FUNCTION_BLOCK FB_autoStore EXTENDS FB_Generic
VAR_INPUT
END_VAR
VAR_OUTPUT
END_VAR
VAR
	lamp			: BOOL;	
	eStates			: E_AutoStore_States := E_AutoStore_States.IDLE;;
	eStateTemp		: E_AutoStore_States := E_AutoStore_States.IDLE;
	
	mcAxis_lift 			: FB_MotionAxis_MC;
	st_mcAxis_lift 			: ST_MotionAxis_MC;
	AxisRef_lift			: AXIS_REF;
	
	mcAxis_transfer 		: FB_MotionAxis_MC;
	st_mcAxis_transfer		: ST_MotionAxis_MC;
	AxisRef_transfer		: AXIS_REF;
	
	door_closed						: BOOL;
	button_start					: BOOL;	
	button_stop						: BOOL;	
	sensor_lift_atDownPos			: BOOL;
	sensor_transfer_atWorkingPos	: BOOL;
	sensor_transfer_atFeedingPos	: BOOL;
	
	bUpStairs						: BOOL;
	bExchangeTote					: BOOL;
	
	
	autostore_status	: AutostoreStatus;
END_VAR	
VAR PERSISTENT
	rPos_lift_up				: REAL;//340
	rPos_lift_down				: REAL;
	rPos_transfer_feeding		: REAL;
	rPos_transfer_working		: REAL;//636	
END_VAR

SUPER^();
IF sInstanceName='autoStore_1' THEN
	rPos_lift_up				:= 350;
	rPos_lift_down				:= 0;
	rPos_transfer_feeding		:= 0;
	rPos_transfer_working		:= 656;	
END_IF
IF sInstanceName='autoStore_2' THEN
	rPos_lift_up				:= 350;
	rPos_lift_down				:= 0;
	rPos_transfer_feeding		:= 0;
	rPos_transfer_working		:= 624;	
END_IF
IF sInstanceName='autoStore_1' THEN
	IF NOT subscribed THEN
		GVL.PubSubService.Subscribe(E_Topics.AUTOSTORE1_EXCHANGE,sInstanceName,THIS^);
		subscribed	:= TRUE;
	END_IF
END_IF
IF sInstanceName='autoStore_2' THEN
	IF NOT subscribed THEN
		GVL.PubSubService.Subscribe(E_Topics.AUTOSTORE2_EXCHANGE,sInstanceName,THIS^);
		subscribed	:= TRUE;
	END_IF
END_IF

//sComponent_name		:= _sInstanceName;
//iComponetID			:= ModuleID.SAMPLE1;

infoLevel	:= ServerityLevelType.WARNING;

(*
Description: 
the callback that will be invoked when there is a publish for what the subscriber was subscribed to.
*)
METHOD Callback
VAR_INPUT
	data : PubSubData;
END_VAR
IF door_closed THEN
	IF sInstanceName='autoStore_1' THEN
		CASE data.Topic OF
			E_Topics.AUTOSTORE1_EXCHANGE:
				IF autostore_status<>AutostoreStatus.EXCHANGING THEN
					bExchangeTote	:= TRUE;	
				END_IF
		END_CASE	
	END_IF
	IF sInstanceName='autoStore_2' THEN
		CASE data.Topic OF
			E_Topics.AUTOSTORE2_EXCHANGE:
				IF autostore_status<>AutostoreStatus.EXCHANGING THEN
					bExchangeTote	:= TRUE;	
				END_IF		
		END_CASE	
	END_IF
END_IF
END_METHOD

{attribute 'object_name' := 'M_Aborting'}
METHOD M_Aborting
CASE fbUnitModeManager.eModeStatus OF	
	ePMLProtUnitMode_Production, ePMLProtUnitMode_Manual:		

		st_mcAxis_lift.mcMoveAbsolute.Execute		:= FALSE;
		st_mcAxis_lift.mcStop.Execute				:= TRUE;	
		st_mcAxis_transfer.mcMoveAbsolute.Execute	:= FALSE;
		st_mcAxis_transfer.mcStop.Execute			:= TRUE;
		iAging_test	:= 0;
		M_StateComplete();
			
	ePMLProtUnitMode_Maintenance, ePMLUnitMode_Service:
		
		M_StateComplete();
END_CASE
END_METHOD

METHOD M_agingTest : BOOL
VAR_INPUT
	rVelocity_percent	: REAL;
END_VAR
END_METHOD

{attribute 'object_name' := 'M_Completing'}
METHOD M_Completing
CASE fbUnitModeManager.eModeStatus OF
	ePMLProtUnitMode_Production:
		;
END_CASE
END_METHOD

{attribute 'object_name' := 'M_Execute'}
METHOD M_Execute
IF door_closed THEN
	st_mcAxis_transfer.mcStop.Execute	:= FALSE;
	st_mcAxis_lift.mcStop.Execute		:= FALSE;
	st_mcAxis_transfer.mcReset.Execute	:= TRUE;
	st_mcAxis_lift.mcReset.Execute		:= TRUE;	
ELSE
	st_mcAxis_transfer.mcStop.Execute	:= TRUE;
	st_mcAxis_lift.mcStop.Execute		:= TRUE;
	RETURN;
END_IF
CASE fbUnitModeManager.eModeStatus OF
	ePMLProtUnitMode_Production:		//Mode Production
//////////////////////////////////////////////////////////timeout//////////////////////////////////////////	
		iStateTemp	:= eStateTemp;
		ton_timeout();
		IF eStateTemp=eStates THEN
			ton_timeout.IN	:=TRUE;
		ELSE
			ton_timeout.IN	:=FALSE;
			eStateTemp	:= eStates;	
			M_Log(eLogType:=ServerityLevelType.INFO,sTextLog:='');
			IF ton_timeout.Q THEN
				RETURN;
			END_IF
		END_IF
		IF ton_timeout.Q THEN	
			ton_timeout.IN	:=FALSE;
			CASE eStates OF	
				E_AutoStore_States.ERROR:	
					alarm_temp.Message	:= GenerateErrorMsg(errorType:='M',iState := iStateTemp,errorMsg:='in error state.');
				ELSE
				alarm_temp.Message	:= GenerateErrorMsg(errorType:='M',iState := iStateTemp,errorMsg:='time out');
			END_CASE
//////////////////////////////////////////////////////////states don't want to timeout and trig error//////////////////////////////////////////				
			IF 	eStates<>E_AutoStore_States.IDLE AND
				eStates<>E_AutoStore_States.WAIT AND
				eStates<>E_AutoStore_States.WAIT_CMD
			THEN 
				IF sInstanceName='autoStore_1' THEN
					GVL.pml_adminAlarm.M_SetAlarm(stAdmin:=GVL.PackTags1.Admin,stAlarm:=alarm_temp);
				END_IF
				IF sInstanceName='autoStore_2' THEN
					GVL.pml_adminAlarm.M_SetAlarm(stAdmin:=GVL.PackTags2.Admin,stAlarm:=alarm_temp);
				END_IF					
			END_IF
		END_IF
//////////////////////////////////////////////////////////auto running process//////////////////////////////////////////			
		CASE eStates OF 
				E_AutoStore_States.IDLE:
					ton_timeout.PT	:= T#1MS;						
					eStates	:= E_AutoStore_States.INIT;				
				E_AutoStore_States.INIT:
					ton_timeout.PT	:= T#1S;
					st_mcAxis_transfer.mcMoveAbsolute.Execute	:= FALSE;
					st_mcAxis_lift.mcMoveAbsolute.Execute	:= FALSE;
					autostore_status	:= AutostoreStatus.UNKNOWN;
					eStates	:= E_AutoStore_States.WAIT; 
				E_AutoStore_States.WAIT:
					ton_timeout.PT	:= T#10S;
					eStates	:= E_AutoStore_States.WAIT_CMD; 
				E_AutoStore_States.WAIT_CMD:
					IF bExchangeTote OR button_start THEN
						bExchangeTote	:= FALSE;
						autostore_status	:= AutostoreStatus.EXCHANGING;
						eStates	:= E_AutoStore_States.LIFT_MOVE_DOWN;
					END_IF
				////////////////////////////lift move down///////////////////////////////////		
				E_AutoStore_States.LIFT_MOVE_DOWN:	
					st_mcAxis_lift.mcMoveAbsolute.Execute	:= TRUE;					
					st_mcAxis_lift.rActualPosSet	:= rPos_lift_down;
					st_mcAxis_lift.rVelocitySet		:= 400;					
					IF st_mcAxis_lift.mcMoveAbsolute.Done THEN
						st_mcAxis_lift.mcMoveAbsolute.Execute	:= FALSE;
						eStates	:= E_AutoStore_States.LIFT_DOWN_SENSOR_DETECTED;
					END_IF
				E_AutoStore_States.LIFT_DOWN_SENSOR_DETECTED:	
					IF TRUE OR sensor_lift_atDownPos THEN
						IF bUpStairs THEN
							eStates	:= E_AutoStore_States.TRANSFER_MOVE_FEEDING;
							bUpStairs	:= FALSE;
						ELSE
							eStates	:= E_AutoStore_States.TRANSFER_MOVE_WORKING;
							bUpStairs	:= TRUE;
						END_IF					
					END_IF
				////////////////////////////upstairs///////////////////////////////////	
				E_AutoStore_States.TRANSFER_MOVE_FEEDING:	
					st_mcAxis_transfer.mcMoveAbsolute.Execute	:= TRUE;					
					st_mcAxis_transfer.rActualPosSet	:= rPos_transfer_feeding;
					st_mcAxis_transfer.rVelocitySet		:= 600;					
					IF st_mcAxis_transfer.mcMoveAbsolute.Done THEN
						st_mcAxis_transfer.mcMoveAbsolute.Execute	:= FALSE;
						eStates	:= E_AutoStore_States.TRANSFER_FEEDING_SENSOR_DETECTED;
					END_IF				

				E_AutoStore_States.TRANSFER_FEEDING_SENSOR_DETECTED:
					IF sensor_transfer_atFeedingPos OR TRUE THEN//todo:add this sensor
						eStates	:= E_AutoStore_States.LIFT_MOVE_UP;
					END_IF									
				////////////////////////////downstairs///////////////////////////////////		
				E_AutoStore_States.TRANSFER_MOVE_WORKING:	
					st_mcAxis_transfer.mcMoveAbsolute.Execute	:= TRUE;					
					st_mcAxis_transfer.rActualPosSet	:= rPos_transfer_working;
					st_mcAxis_transfer.rVelocitySet		:= 600;					
					IF st_mcAxis_transfer.mcMoveAbsolute.Done THEN
						st_mcAxis_transfer.mcMoveAbsolute.Execute	:= FALSE;
						eStates	:= E_AutoStore_States.TRANSFER_WORKING_SENSOR_DETECTED;
					END_IF					
				E_AutoStore_States.TRANSFER_WORKING_SENSOR_DETECTED:
					IF sensor_transfer_atWorkingPos OR TRUE THEN//todo:adjust the position
						eStates	:= E_AutoStore_States.LIFT_MOVE_UP;
					END_IF
					
				////////////////////////////lift move up///////////////////////////////////	
				E_AutoStore_States.LIFT_MOVE_UP:
					st_mcAxis_lift.mcMoveAbsolute.Execute	:= TRUE;					
					st_mcAxis_lift.rActualPosSet	:= rPos_lift_up;
					st_mcAxis_lift.rVelocitySet		:= 150;					
					IF st_mcAxis_lift.mcMoveAbsolute.Done THEN
						st_mcAxis_lift.mcMoveAbsolute.Execute	:= FALSE;
						eStates	:= E_AutoStore_States.DONE;
					END_IF		

				
				E_AutoStore_States.DONE:
					autostore_status	:= AutostoreStatus.READY;
					eStates	:= E_AutoStore_States.WAIT_CMD;
				E_AutoStore_States.ERROR:
					;
			END_CASE
		
		
	ePMLProtUnitMode_Maintenance, ePMLUnitMode_Service:		
		//
		
	ePMLProtUnitMode_Manual:		//Manaul

END_CASE
END_METHOD

{attribute 'object_name' := 'M_Holding'}
METHOD M_Holding
CASE fbUnitModeManager.eModeStatus OF
	ePMLProtUnitMode_Production:		//Mode Production
		//Finisch the actual seperationstep	
		

	ePMLProtUnitMode_Maintenance:
		M_StateComplete();
END_CASE
END_METHOD

{attribute 'object_name' := 'M_Idle'}
METHOD M_Idle
IF G_HMI.bAging_test THEN
	//M_agingTest();
END_IF
END_METHOD

METHOD M_mapping : BOOL
VAR_INPUT
END_VAR
IF sInstanceName='autoStore_1' THEN	
	(****************************digital input***************************************************)
	st_mcAxis_lift.limit_sensor_positive		:= 	arDI[20].Ch[0] ;
	st_mcAxis_lift.limit_sensor_negative		:= 	arDI[20].Ch[1] ;
	door_closed									:= 	arDI[20].Ch[2] ;
	button_start								:= 	arDI[20].Ch[3] ;
	button_stop									:= 	arDI[20].Ch[4] ;
	sensor_lift_atDownPos						:= 	arDI[20].Ch[5] ;
	st_mcAxis_transfer.limit_sensor_positive	:= 	arDI[20].Ch[6] ;
	st_mcAxis_transfer.limit_sensor_negative	:= 	arDI[20].Ch[7] ;	
	sensor_transfer_atWorkingPos				:= 	arDI[20].Ch[8] ;	
//	sensor_transfer_atFeedingPos				:= 	arDI[20].Ch[9] ;	
		

	/////////////////////////////////////axis config////////////////////////////////////////
	mcAxis_transfer
	(
		ZSN		:=  TRUE OR (st_mcAxis_transfer.limit_sensor_negative (*AND sensor_lift_atDownPos*)) OR st_mcAxis_transfer.xHoming, //TODO link to digital input
		ZSP		:=  TRUE OR (st_mcAxis_transfer.limit_sensor_positive (*AND sensor_lift_atDownPos*)) OR st_mcAxis_transfer.xHoming, //TODO link to digital input
		IN_OUT	:= st_mcAxis_transfer	, 
		AXIS	:= AxisRef_transfer	, 
	);
	st_mcAxis_transfer.bPosSensorShow	:= TRUE;
	st_mcAxis_transfer.bNegSensorShow	:= TRUE;
	st_mcAxis_transfer.bStopButtonShow	:= TRUE;
	st_mcAxis_transfer.rMaxAcceleration	:= 50000;
	st_mcAxis_transfer.rMaxDeceleration	:= 50000;
	st_mcAxis_transfer.rMaxJerk			:= 500000;
	st_mcAxis_transfer.rAcceleration	:= 2500;
	st_mcAxis_transfer.rDeceleration	:= 2500;
	st_mcAxis_transfer.rJerk			:= 12500;
	st_mcAxis_transfer.rMaxVelocity		:= 100;
	st_mcAxis_transfer.rMaxDistance		:= 50;
	st_mcAxis_transfer.bPosSen	:=  st_mcAxis_transfer.limit_sensor_positive ;//TODO link to digital input
	st_mcAxis_transfer.bNegSen	:=  st_mcAxis_transfer.limit_sensor_negative ;//TODO link to digital input
	st_mcAxis_transfer.mcHome.bCalibrationCam	:= TRUE;//TODO link to digital input origin
	st_mcAxis_transfer.bPositionSensor	:= TRUE;//TODO link to digital input origin
	st_mcAxis_transfer.bdirFW	:= TRUE;
	st_mcAxis_transfer.sNetID := '192.168.11.159.8.1';
	st_mcAxis_transfer.nSlaveAddr	:= 1004;
	st_mcAxis_transfer.rToqueLimitSet	:= 80;	
	
	mcAxis_lift
	(
		ZSN		:=   TRUE OR st_mcAxis_lift.limit_sensor_negative  OR st_mcAxis_lift.xHoming, //TODO link to digital input
		ZSP		:=   TRUE OR (st_mcAxis_lift.limit_sensor_positive (*AND sensor_transfer_atWorkingPos*))  OR st_mcAxis_lift.xHoming, //TODO link to digital input
		IN_OUT	:= st_mcAxis_lift	, 
		AXIS	:= AxisRef_lift	, 
	);
	st_mcAxis_lift.bPosSensorShow	:= TRUE;
	st_mcAxis_lift.bNegSensorShow	:= TRUE;
	st_mcAxis_lift.bStopButtonShow	:= TRUE;
	st_mcAxis_lift.rMaxAcceleration	:= 50000;
	st_mcAxis_lift.rMaxDeceleration	:= 50000;
	st_mcAxis_lift.rMaxJerk			:= 500000;
	st_mcAxis_lift.rAcceleration	:= 2500;
	st_mcAxis_lift.rDeceleration	:= 2500;
	st_mcAxis_lift.rJerk			:= 12500;
	st_mcAxis_lift.rMaxVelocity		:= 100;
	st_mcAxis_lift.rMaxDistance		:= 50;
	st_mcAxis_lift.bPosSen	:=  st_mcAxis_lift.limit_sensor_positive ;//TODO link to digital input
	st_mcAxis_lift.bNegSen	:=  TRUE(*st_mcAxis_lift.limit_sensor_negative*) ;//TODO link to digital input
	st_mcAxis_lift.mcHome.bCalibrationCam	:= TRUE;//TODO link to digital input origin
	st_mcAxis_lift.bPositionSensor	:= TRUE;//TODO link to digital input origin
	st_mcAxis_lift.bdirFW	:= TRUE;
	st_mcAxis_lift.sNetID := '192.168.11.159.8.1';
	st_mcAxis_lift.nSlaveAddr	:= 1005;
	st_mcAxis_lift.rToqueLimitSet	:= 80;
END_IF




IF sInstanceName='autoStore_2' THEN	
	(****************************digital input***************************************************)
	st_mcAxis_lift.limit_sensor_positive		:= 	arDI[21].Ch[0] ;
	st_mcAxis_lift.limit_sensor_negative		:= 	arDI[21].Ch[1] ;
	door_closed									:= 	arDI[21].Ch[2] ;
	button_start								:= 	arDI[21].Ch[3] ;
	button_stop									:= 	arDI[21].Ch[4] ;
	sensor_lift_atDownPos						:= 	arDI[21].Ch[5] ;
	st_mcAxis_transfer.limit_sensor_positive	:= 	arDI[21].Ch[6] ;
	st_mcAxis_transfer.limit_sensor_negative	:= 	arDI[21].Ch[7] ;	
	sensor_transfer_atWorkingPos				:= 	arDI[21].Ch[8] ;	
//	sensor_transfer_atFeedingPos				:= 	arDI[21].Ch[9] ;	
		

	/////////////////////////////////////axis config////////////////////////////////////////
	mcAxis_transfer
	(
		ZSN		:=  TRUE OR (st_mcAxis_transfer.limit_sensor_negative (*AND sensor_lift_atDownPos*)) OR st_mcAxis_transfer.xHoming, //TODO link to digital input
		ZSP		:=  TRUE OR (st_mcAxis_transfer.limit_sensor_positive (*AND sensor_lift_atDownPos*)) OR st_mcAxis_transfer.xHoming, //TODO link to digital input
		IN_OUT	:= st_mcAxis_transfer	, 
		AXIS	:= AxisRef_transfer	, 
	);
	st_mcAxis_transfer.bPosSensorShow	:= TRUE;
	st_mcAxis_transfer.bNegSensorShow	:= TRUE;
	st_mcAxis_transfer.bStopButtonShow	:= TRUE;
	st_mcAxis_transfer.rMaxAcceleration	:= 50000;
	st_mcAxis_transfer.rMaxDeceleration	:= 50000;
	st_mcAxis_transfer.rMaxJerk			:= 500000;
	st_mcAxis_transfer.rAcceleration	:= 2500;
	st_mcAxis_transfer.rDeceleration	:= 2500;
	st_mcAxis_transfer.rJerk			:= 12500;
	st_mcAxis_transfer.rMaxVelocity		:= 100;
	st_mcAxis_transfer.rMaxDistance		:= 50;
	st_mcAxis_transfer.bPosSen	:=  st_mcAxis_transfer.limit_sensor_positive ;//TODO link to digital input
	st_mcAxis_transfer.bNegSen	:=  st_mcAxis_transfer.limit_sensor_negative ;//TODO link to digital input
	st_mcAxis_transfer.mcHome.bCalibrationCam	:= TRUE;//TODO link to digital input origin
	st_mcAxis_transfer.bPositionSensor	:= TRUE;//TODO link to digital input origin
	st_mcAxis_transfer.bdirFW	:= TRUE;
	st_mcAxis_transfer.sNetID := '192.168.11.159.10.1';
	st_mcAxis_transfer.nSlaveAddr	:= 1004;
	st_mcAxis_transfer.rToqueLimitSet	:= 80;	
	
	mcAxis_lift
	(
		ZSN		:=   TRUE OR st_mcAxis_lift.limit_sensor_negative  OR st_mcAxis_lift.xHoming, //TODO link to digital input
		ZSP		:=   TRUE OR (st_mcAxis_lift.limit_sensor_positive (*AND sensor_transfer_atWorkingPos*))  OR st_mcAxis_lift.xHoming, //TODO link to digital input
		IN_OUT	:= st_mcAxis_lift	, 
		AXIS	:= AxisRef_lift	, 
	);
	st_mcAxis_lift.bPosSensorShow	:= TRUE;
	st_mcAxis_lift.bNegSensorShow	:= TRUE;
	st_mcAxis_lift.bStopButtonShow	:= TRUE;
	st_mcAxis_lift.rMaxAcceleration	:= 50000;
	st_mcAxis_lift.rMaxDeceleration	:= 50000;
	st_mcAxis_lift.rMaxJerk			:= 500000;
	st_mcAxis_lift.rAcceleration	:= 2500;
	st_mcAxis_lift.rDeceleration	:= 2500;
	st_mcAxis_lift.rJerk			:= 12500;
	st_mcAxis_lift.rMaxVelocity		:= 100;
	st_mcAxis_lift.rMaxDistance		:= 50;
	st_mcAxis_lift.bPosSen	:=  st_mcAxis_lift.limit_sensor_positive ;//TODO link to digital input
	st_mcAxis_lift.bNegSen	:=  TRUE(*st_mcAxis_lift.limit_sensor_negative*) ;//TODO link to digital input
	st_mcAxis_lift.mcHome.bCalibrationCam	:= TRUE;//TODO link to digital input origin
	st_mcAxis_lift.bPositionSensor	:= TRUE;//TODO link to digital input origin
	st_mcAxis_lift.bdirFW	:= TRUE;
	st_mcAxis_lift.sNetID := '192.168.11.159.10.1';
	st_mcAxis_lift.nSlaveAddr	:= 1005;
	st_mcAxis_lift.rToqueLimitSet	:= 80;
END_IF
END_METHOD

METHOD M_Reset
VAR_INPUT
END_VAR
//Take away all commands
IF GVL.stChangeIntoProduction.bYesReset THEN
;
END_IF
END_METHOD

{attribute 'object_name' := 'M_Resetting'}
METHOD M_Resetting
CASE fbUnitModeManager.eModeStatus OF
	ePMLProtUnitMode_Production:		//Production, Mantainance, Manual
		lamp	:= FALSE;
		eStates :=E_SampleStates.IDLE;
		M_StateComplete();
	
	ePMLProtUnitMode_Maintenance, ePMLProtUnitMode_Manual, ePMLUnitMode_Service:
		M_StateComplete();
END_CASE
END_METHOD

{attribute 'object_name' := 'M_Starting'}
METHOD M_Starting
CASE fbUnitModeManager.eModeStatus OF
	ePMLProtUnitMode_Production:		//Production, Mantainance, Manual
		st_mcAxis_transfer.mcPower.Enable	:= TRUE;
		st_mcAxis_lift.mcPower.Enable	:= TRUE;
		IF st_mcAxis_transfer.mcPower.Status AND st_mcAxis_lift.mcPower.Status THEN
			eStates	:= E_AutoStore_States.IDLE;	
			M_StateComplete();
		END_IF
		
	ePMLProtUnitMode_Maintenance, ePMLProtUnitMode_Manual, ePMLUnitMode_Service:
		M_StateComplete();
END_CASE
END_METHOD

{attribute 'object_name' := 'M_Stopping'}
METHOD M_Stopping

CASE fbUnitModeManager.eModeStatus OF
	ePMLProtUnitMode_Production:		//Mode Production
//////////////////////////////////////////////////////////timeout//////////////////////////////////////////	
		iStateTemp	:= eStateTemp;
		ton_timeout();
		IF eStateTemp=eStates THEN
			ton_timeout.IN	:=TRUE;
		ELSE
			ton_timeout.IN	:=FALSE;
			eStateTemp	:= eStates;	
			M_Log(eLogType:=ServerityLevelType.INFO,sTextLog:='');
			IF ton_timeout.Q THEN
				RETURN;
			END_IF
		END_IF
		IF ton_timeout.Q THEN	
			ton_timeout.IN	:=FALSE;
			CASE eStates OF	
				E_AutoStore_States.ERROR:	
					alarm_temp.Message	:= GenerateErrorMsg(errorType:='M',iState := iStateTemp,errorMsg:='in error state.');
				ELSE
				alarm_temp.Message	:= GenerateErrorMsg(errorType:='M',iState := iStateTemp,errorMsg:='time out');
			END_CASE
//////////////////////////////////////////////////////////states don't want to timeout and trig error//////////////////////////////////////////				
			IF 	eStates<>E_AutoStore_States.IDLE AND
				eStates<>E_AutoStore_States.WAIT AND
				eStates<>E_AutoStore_States.WAIT_CMD
			THEN 
				IF sInstanceName='autoStore_1' THEN
					GVL.pml_adminAlarm.M_SetAlarm(stAdmin:=GVL.PackTags1.Admin,stAlarm:=alarm_temp);
				END_IF
				IF sInstanceName='autoStore_2' THEN
					GVL.pml_adminAlarm.M_SetAlarm(stAdmin:=GVL.PackTags2.Admin,stAlarm:=alarm_temp);
				END_IF					
			END_IF
		END_IF
//////////////////////////////////////////////////////////auto running process//////////////////////////////////////////			
		CASE eStates OF 
				E_AutoStore_States.IDLE:
					ton_timeout.PT	:= T#1MS;						
					eStates	:= E_AutoStore_States.INIT;				
				E_AutoStore_States.INIT:
					ton_timeout.PT	:= T#1S;
					eStates	:= E_AutoStore_States.WAIT; 
				E_AutoStore_States.WAIT:
					ton_timeout.PT	:= T#10S;
					eStates	:= E_AutoStore_States.WAIT_CMD; 
				E_AutoStore_States.WAIT_CMD:
					M_StateComplete();
					IF bExchangeTote THEN
						bExchangeTote	:= FALSE;
						eStates	:= E_AutoStore_States.LIFT_MOVE_DOWN;
					END_IF
				////////////////////////////lift move down///////////////////////////////////		
				E_AutoStore_States.LIFT_MOVE_DOWN:	
					st_mcAxis_lift.mcMoveAbsolute.Execute	:= TRUE;					
					st_mcAxis_lift.rActualPosSet	:= rPos_lift_down;
					st_mcAxis_lift.rVelocitySet		:= 100;					
					IF st_mcAxis_lift.mcMoveAbsolute.Done THEN
						eStates	:= E_AutoStore_States.LIFT_DOWN_SENSOR_DETECTED;
					END_IF
				E_AutoStore_States.LIFT_DOWN_SENSOR_DETECTED:	
					IF sensor_lift_atDownPos THEN
						IF bUpStairs THEN
							eStates	:= E_AutoStore_States.TRANSFER_MOVE_FEEDING;
							bUpStairs	:= FALSE;
						ELSE
							eStates	:= E_AutoStore_States.TRANSFER_MOVE_WORKING;
							bUpStairs	:= TRUE;
						END_IF					
					END_IF
				////////////////////////////upstairs///////////////////////////////////	
				E_AutoStore_States.TRANSFER_MOVE_FEEDING:	
					st_mcAxis_transfer.mcMoveAbsolute.Execute	:= TRUE;					
					st_mcAxis_transfer.rActualPosSet	:= rPos_transfer_feeding;
					st_mcAxis_transfer.rVelocitySet		:= 100;					
					IF st_mcAxis_transfer.mcMoveAbsolute.Done THEN
						eStates	:= E_AutoStore_States.TRANSFER_FEEDING_SENSOR_DETECTED;
					END_IF				

				E_AutoStore_States.TRANSFER_FEEDING_SENSOR_DETECTED:
					IF sensor_transfer_atFeedingPos OR TRUE THEN//todo:add this sensor
						eStates	:= E_AutoStore_States.LIFT_MOVE_UP;
					END_IF									
				////////////////////////////downstairs///////////////////////////////////		
				E_AutoStore_States.TRANSFER_MOVE_WORKING:	
					st_mcAxis_transfer.mcMoveAbsolute.Execute	:= TRUE;					
					st_mcAxis_transfer.rActualPosSet	:= rPos_transfer_working;
					st_mcAxis_transfer.rVelocitySet		:= 100;					
					IF st_mcAxis_transfer.mcMoveAbsolute.Done THEN
						eStates	:= E_AutoStore_States.TRANSFER_WORKING_SENSOR_DETECTED;
					END_IF					
				E_AutoStore_States.TRANSFER_WORKING_SENSOR_DETECTED:
					IF sensor_transfer_atWorkingPos THEN
						eStates	:= E_AutoStore_States.LIFT_MOVE_UP;
					END_IF
					
				////////////////////////////lift move up///////////////////////////////////	
				E_AutoStore_States.LIFT_MOVE_UP:
					st_mcAxis_lift.mcMoveAbsolute.Execute	:= TRUE;					
					st_mcAxis_lift.rActualPosSet	:= rPos_lift_up;
					st_mcAxis_lift.rVelocitySet		:= 100;					
					IF st_mcAxis_lift.mcMoveAbsolute.Done THEN
						eStates	:= E_AutoStore_States.DONE;
					END_IF		

				
				E_AutoStore_States.DONE:
					eStates	:= E_AutoStore_States.IDLE;
					M_StateComplete();
				E_AutoStore_States.ERROR:
					;
			END_CASE
		
		
	ePMLProtUnitMode_Maintenance, ePMLUnitMode_Service:		
		//
		
	ePMLProtUnitMode_Manual:		//Manaul

END_CASE
END_METHOD

{attribute 'object_name' := 'M_Undefined'}
METHOD M_Undefined

bUndefinedDone					:= TRUE;
END_METHOD

METHOD ParseStateToString : STRING
VAR_INPUT
END_VAR
CASE THIS^.eStates OF
	E_AutoStore_States.IDLE:
		ParseStateToString	:='IDLE';
	E_AutoStore_States.INIT:
		ParseStateToString	:='INIT';
	E_AutoStore_States.CHECK:
		ParseStateToString	:='CHECK';

	E_AutoStore_States.WAIT:
		ParseStateToString	:='WAIT';

	E_AutoStore_States.DONE:	
		ParseStateToString	:='DONE';
	E_AutoStore_States.ERROR:
		ParseStateToString	:='ERROR';
	ELSE
		ParseStateToString	:='UNKNOW STATE';
END_CASE
END_METHOD

END_FUNCTION_BLOCK

(* stored: Version 1.1.0.1, ProductVersion 3.1.4024.12
   POU FB_autoStore: Id {928a0155-c36c-415e-9368-ea4c51d98670}, SpecialFunc None
   Method Callback: Id {a6bbd39f-2150-4ac8-bd46-3426611ab3aa}
   Method M_Aborting: Id {43d30a98-ba2d-4ee3-a388-632bc0ec3cf0}
   Method M_agingTest: Id {586b505d-8f43-40e1-8ab9-a036d9d23d49}
   Method M_Completing: Id {05e8a900-f003-4d6c-b3a8-567bb1951b3a}
   Method M_Execute: Id {6f10dd64-04f0-4b2a-8681-455f4d918556}
   Method M_Holding: Id {9f18e7fa-a28d-4512-ac0f-c8ef5c3137ca}
   Method M_Idle: Id {02d44905-2bed-4a37-9a21-0d818428d446}
   Method M_mapping: Id {fe3409f9-2642-4d57-8c0c-03b05bca0fc4}
   Method M_Reset: Id {4f94f8a4-a16d-43ea-b0f0-409e3aade142}
   Method M_Resetting: Id {51654668-1d9f-43f1-be34-eaae0b34b683}
   Method M_Starting: Id {6bf2a7b8-ba0a-443d-9bd9-157b795c08a2}
   Method M_Stopping: Id {f43f7b4b-ef4e-433f-a431-82b654dcfe16}
   Method M_Undefined: Id {1523c926-ded0-4f2e-8d47-c558e8648371}
   Method ParseStateToString: Id {29842482-7149-4ae9-b12c-8be8de69ff66} *)
